# EPICS IOC start-up script: iocs/zaberMotionIOC/iocBoot/iocZaberMotion/common.iocsh
< envPaths

cd "${TOP}"

## Register all support components
dbLoadDatabase "dbd/zaberMotion.dbd"
zaberMotion_registerRecordDeviceDriver pdbbase

## motorUtil (allstop & alldone)
dbLoadRecords("$(MOTOR)/db/motorUtil.db", "P=zaberMotion:")

cd "${TOP}/iocBoot/${IOC}"

##
< dbPath.cmd.zaber
< motor.cmd.zaber
< profile.cmd.zaber

iocInit

## motorUtil (allstop & alldone)
motorUtilInit("zaberMotion:")

# Boot complete
